// TIA Portal V20 export
// export: Created 2025-12-01T14:56:59.921487Z, ExportSetting None, DisplayName Totally Integrated Automation Portal, DisplayVersion V20 Update 3, DisplayName TIA Portal Openness, DisplayVersion V20 Update 3, DisplayName TIA Portal Version Control Interface, DisplayVersion V20 Update 3, DisplayName STEP 7 Professional, DisplayVersion V20 Update 3, DisplayName STEP 7 Safety, DisplayVersion V20 Update 2, DisplayName WinCC Basic/Comfort/Advanced, DisplayVersion V20 Update 3, DisplayName WinCC Professional, DisplayVersion V20 Update 3, DisplayName WinCC Unified, DisplayVersion V20 Update 3
FUNCTION "FC425_TL_Sep_Salida" : Void   // FC425, LAD
{ S7_Optimized_Access := 'FALSE' }
AUTHOR : TLigero
NAME : 20190131
VERSION : 3.3
// ////////////////////////////
// Modificada 27-11-2012
// Separación salida entre culo de primera caja y cara de la segunda para distanci 
// kte mayor flujo con tamaños diferentes de cajas
// ////////////////////////////
// stored: AutoNumber false, SetENOAutomatically false
   VAR_INPUT
      Mesa : UInt;
      En_Tension : Bool;
      PhsMx : Bool;
      Termico_Tx : Bool;
      Avance_Tx : Bool;
      Modo_Pasoapaso_Tx : Bool;
      AVTF_MAnt_Mx : Bool;
      PTF_Mx_MSig : Bool;
      NXT_Avance : Bool;
      V_CNT_pHsMx : UDInt;
      V_Paro : UDInt;
      V_Separacion : UDInt;
      V_Caja_Max : UDInt;
      V_TOut_Tx_Mx : UDInt;
      V_Acumulacion : UDInt;
   END_VAR
   VAR_OUTPUT
      PTF_MAnt_Mx : Bool;
      AVTF_Mx_MSig : Bool;
   END_VAR
   VAR_IN_OUT
      NXT_Descarga_Act : Bool;
      Carga_Activa_Tx : Bool;
      MAUX_FN_AVTF : Bool;
      Mem_CNT_Tmp_PRES : Bool;
      Mem_CNT_Tmp_Paro_Tx : Bool;
      Mem_CNT_Acumulacion : Bool;
   END_VAR
   VAR_TEMP
      CNT_Sep : Word;
      CNT_Sep_Int : Int;
      CNT_Sep_FORZ_Sep : Int;
      Aux_Parar : Bool;
      Mem_CNT_Separacion : Bool;
      ok_tension : Bool;
      mem_atasco : Bool;
   END_VAR
   VAR_TEMP   // added for the SCL form of the ladder/FBD networks
      _w1 : Bool;
   END_VAR
BEGIN

REGION Network 1: Marca General Error
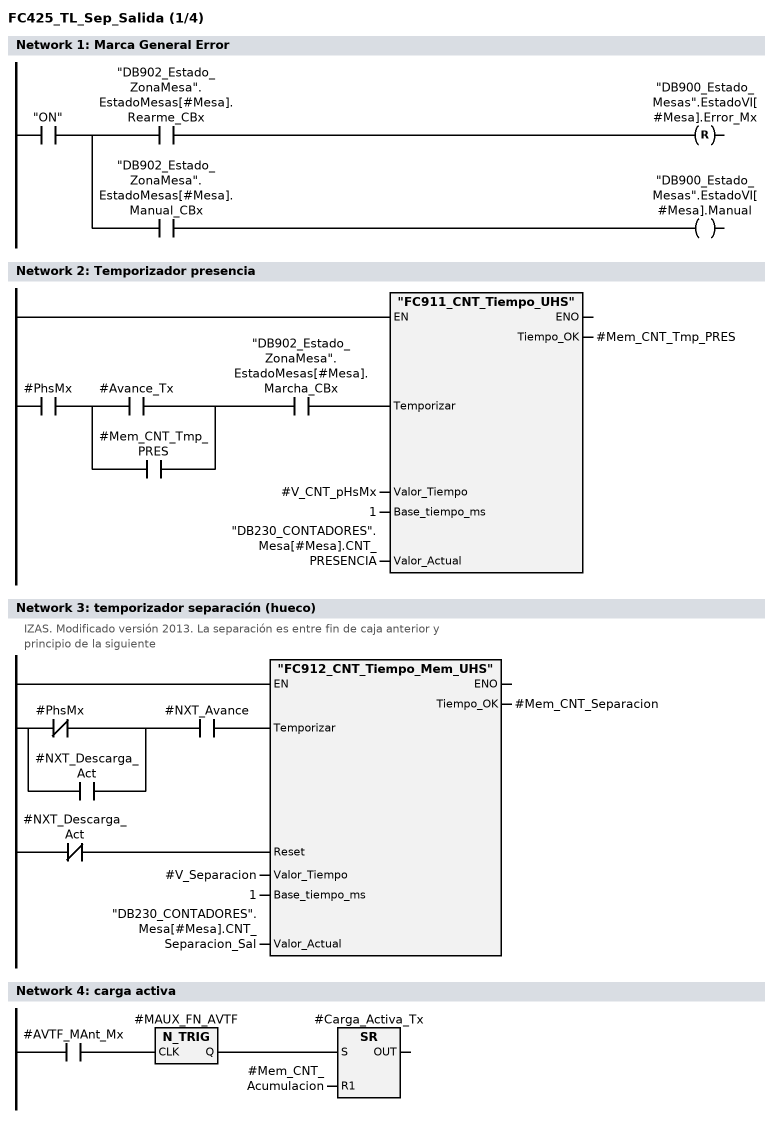
   RUNG wire#powerrail
      Contact( "ON" )
      wire#w1
      Contact( "DB902_Estado_ZonaMesa".EstadoMesas[#Mesa].Rearme_CBx )
      R_Coil( "DB900_Estado_Mesas".EstadoVI[#Mesa].Error_Mx )
   END_RUNG
   RUNG wire#w1
      Contact( "DB902_Estado_ZonaMesa".EstadoMesas[#Mesa].Manual_CBx )
      Coil( "DB900_Estado_Mesas".EstadoVI[#Mesa].Manual )
   END_RUNG
   // the same network as SCL:
   IF "ON" AND "DB902_Estado_ZonaMesa".EstadoMesas[#Mesa].Rearme_CBx THEN
       "DB900_Estado_Mesas".EstadoVI[#Mesa].Error_Mx := FALSE;
   END_IF;
   "DB900_Estado_Mesas".EstadoVI[#Mesa].Manual := "ON" AND "DB902_Estado_ZonaMesa".EstadoMesas[#Mesa].Manual_CBx;
END_REGION

REGION Network 2: Temporizador presencia
   RUNG wire#powerrail
      "FC911_CNT_Tiempo_UHS"(Temporizar := wire#w3, Valor_Tiempo := #V_CNT_pHsMx, Base_tiempo_ms := 1, Valor_Actual := "DB230_CONTADORES".Mesa[#Mesa].CNT_PRESENCIA, Tiempo_OK => #Mem_CNT_Tmp_PRES)
   END_RUNG
   RUNG wire#powerrail
      Contact( #PhsMx )
      wire#w1
      Contact( #Avance_Tx )
      wire#w2
      Contact( "DB902_Estado_ZonaMesa".EstadoMesas[#Mesa].Marcha_CBx )
   END_RUNG wire#w3
   RUNG wire#w1
      Contact( #Mem_CNT_Tmp_PRES )
   END_RUNG wire#w2
   // the same network as SCL:
   "FC911_CNT_Tiempo_UHS"(Temporizar := #PhsMx AND (#Avance_Tx OR #Mem_CNT_Tmp_PRES) AND "DB902_Estado_ZonaMesa".EstadoMesas[#Mesa].Marcha_CBx,
                          Valor_Tiempo := #V_CNT_pHsMx,
                          Base_tiempo_ms := 1,
                          Valor_Actual := "DB230_CONTADORES".Mesa[#Mesa].CNT_PRESENCIA,
                          Tiempo_OK => #Mem_CNT_Tmp_PRES);
END_REGION

REGION Network 3: temporizador separación (hueco)
   // IZAS. Modificado versión 2013. La separación es entre fin de caja anterior y 
   // principio de la siguiente
   RUNG wire#powerrail
      "FC912_CNT_Tiempo_Mem_UHS"(Temporizar := wire#w2, Reset := wire#w3, Valor_Tiempo := #V_Separacion, Base_tiempo_ms := 1, Valor_Actual := "DB230_CONTADORES".Mesa[#Mesa].CNT_Separacion_Sal, Tiempo_OK => #Mem_CNT_Separacion)
   END_RUNG
   RUNG wire#powerrail
      I_Contact( #PhsMx )
      wire#w1
      Contact( #NXT_Avance )
   END_RUNG wire#w2
   RUNG wire#powerrail
      Contact( #NXT_Descarga_Act )
   END_RUNG wire#w1
   RUNG wire#powerrail
      I_Contact( #NXT_Descarga_Act )
   END_RUNG wire#w3
   // the same network as SCL:
   "FC912_CNT_Tiempo_Mem_UHS"(Temporizar := (NOT #PhsMx OR #NXT_Descarga_Act) AND #NXT_Avance,
                           Reset := NOT #NXT_Descarga_Act,
                           Valor_Tiempo := #V_Separacion,
                           Base_tiempo_ms := 1,
                           Valor_Actual := "DB230_CONTADORES".Mesa[#Mesa].CNT_Separacion_Sal,
                           Tiempo_OK => #Mem_CNT_Separacion);
END_REGION

REGION Network 4: carga activa
   RUNG wire#powerrail
      Contact( #AVTF_MAnt_Mx )
      N_Trig( #MAUX_FN_AVTF )
      S_SR(operand := #Carga_Activa_Tx, r1 := #Mem_CNT_Acumulacion)
   END_RUNG
   // the same network as SCL:
   #_w1 := NOT #AVTF_MAnt_Mx AND #MAUX_FN_AVTF;   // falling edge
   #MAUX_FN_AVTF := #AVTF_MAnt_Mx;
   IF #_w1 THEN
       #Carga_Activa_Tx := TRUE;   // SR flip-flop
   END_IF;
   IF #Mem_CNT_Acumulacion THEN #Carga_Activa_Tx := FALSE; END_IF;
END_REGION

REGION Network 5: Temporizador acumulacion
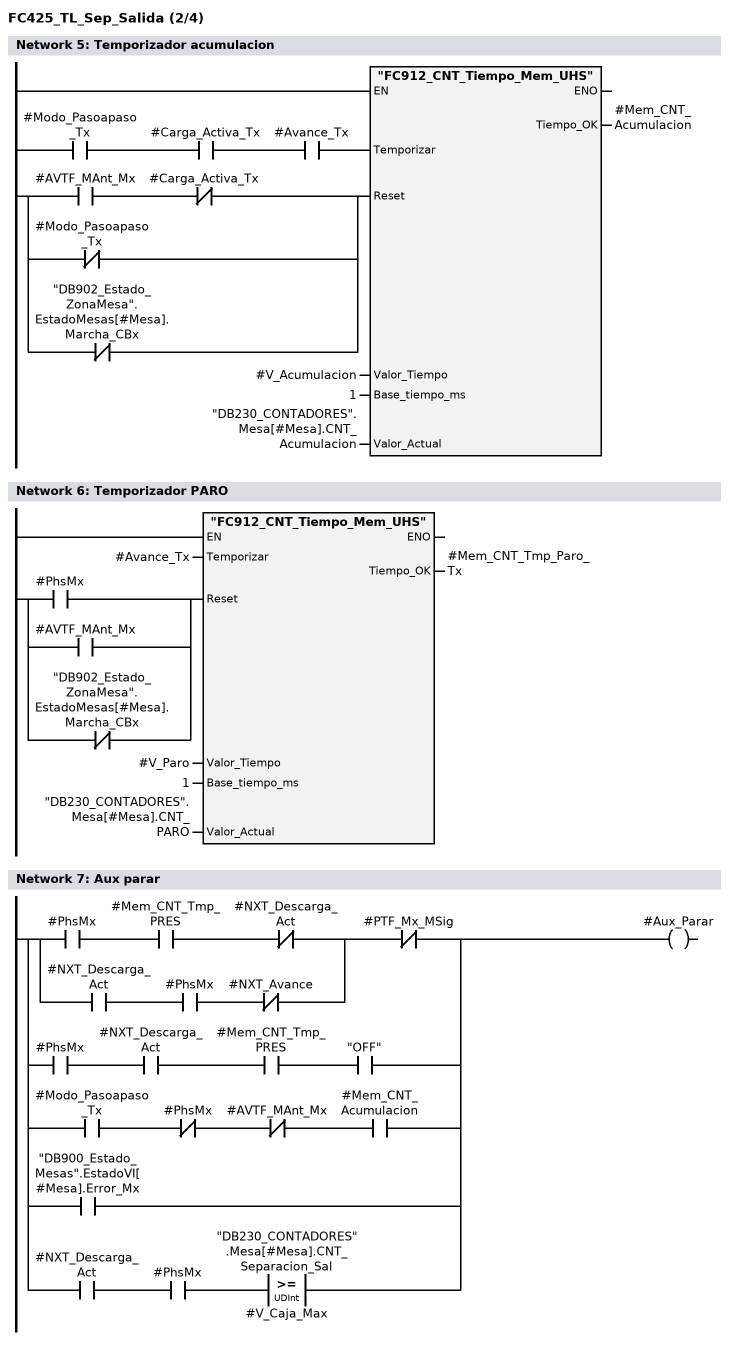
   RUNG wire#powerrail
      "FC912_CNT_Tiempo_Mem_UHS"(Temporizar := wire#w1, Reset := wire#w2, Valor_Tiempo := #V_Acumulacion, Base_tiempo_ms := 1, Valor_Actual := "DB230_CONTADORES".Mesa[#Mesa].CNT_Acumulacion, Tiempo_OK => #Mem_CNT_Acumulacion)
   END_RUNG
   RUNG wire#powerrail
      Contact( #Modo_Pasoapaso_Tx )
      Contact( #Carga_Activa_Tx )
      Contact( #Avance_Tx )
   END_RUNG wire#w1
   RUNG wire#powerrail
      Contact( #AVTF_MAnt_Mx )
      I_Contact( #Carga_Activa_Tx )
   END_RUNG wire#w2
   RUNG wire#powerrail
      I_Contact( #Modo_Pasoapaso_Tx )
   END_RUNG wire#w2
   RUNG wire#powerrail
      I_Contact( "DB902_Estado_ZonaMesa".EstadoMesas[#Mesa].Marcha_CBx )
   END_RUNG wire#w2
   // the same network as SCL:
   "FC912_CNT_Tiempo_Mem_UHS"(Temporizar := #Modo_Pasoapaso_Tx AND #Carga_Activa_Tx AND #Avance_Tx,
                           Reset := (#AVTF_MAnt_Mx AND NOT #Carga_Activa_Tx) OR NOT #Modo_Pasoapaso_Tx OR NOT "DB902_Estado_ZonaMesa".EstadoMesas[#Mesa].Marcha_CBx,
                           Valor_Tiempo := #V_Acumulacion,
                           Base_tiempo_ms := 1,
                           Valor_Actual := "DB230_CONTADORES".Mesa[#Mesa].CNT_Acumulacion,
                           Tiempo_OK => #Mem_CNT_Acumulacion);
END_REGION

REGION Network 6: Temporizador PARO
   RUNG wire#powerrail
      "FC912_CNT_Tiempo_Mem_UHS"(Reset := wire#w1, Temporizar := #Avance_Tx, Valor_Tiempo := #V_Paro, Base_tiempo_ms := 1, Valor_Actual := "DB230_CONTADORES".Mesa[#Mesa].CNT_PARO, Tiempo_OK => #Mem_CNT_Tmp_Paro_Tx)
   END_RUNG
   RUNG wire#powerrail
      Contact( #PhsMx )
   END_RUNG wire#w1
   RUNG wire#powerrail
      Contact( #AVTF_MAnt_Mx )
   END_RUNG wire#w1
   RUNG wire#powerrail
      I_Contact( "DB902_Estado_ZonaMesa".EstadoMesas[#Mesa].Marcha_CBx )
   END_RUNG wire#w1
   // the same network as SCL:
   "FC912_CNT_Tiempo_Mem_UHS"(Temporizar := #Avance_Tx,
                           Reset := #PhsMx OR #AVTF_MAnt_Mx OR NOT "DB902_Estado_ZonaMesa".EstadoMesas[#Mesa].Marcha_CBx,
                           Valor_Tiempo := #V_Paro,
                           Base_tiempo_ms := 1,
                           Valor_Actual := "DB230_CONTADORES".Mesa[#Mesa].CNT_PARO,
                           Tiempo_OK => #Mem_CNT_Tmp_Paro_Tx);
END_REGION

REGION Network 7: Aux parar
   RUNG wire#powerrail
      Contact( #PhsMx )
      Contact( #Mem_CNT_Tmp_PRES )
      I_Contact( #NXT_Descarga_Act )
      wire#w1
      I_Contact( #PTF_Mx_MSig )
      wire#w2
      Coil( #Aux_Parar )
   END_RUNG
   RUNG wire#powerrail
      Contact( #NXT_Descarga_Act )
      Contact( #PhsMx )
      I_Contact( #NXT_Avance )
   END_RUNG wire#w1
   RUNG wire#powerrail
      Contact( #PhsMx )
      Contact( #NXT_Descarga_Act )
      Contact( #Mem_CNT_Tmp_PRES )
      Contact( "OFF" )
   END_RUNG wire#w2
   RUNG wire#powerrail
      Contact( #Modo_Pasoapaso_Tx )
      I_Contact( #PhsMx )
      I_Contact( #AVTF_MAnt_Mx )
      Contact( #Mem_CNT_Acumulacion )
   END_RUNG wire#w2
   RUNG wire#powerrail
      Contact( "DB900_Estado_Mesas".EstadoVI[#Mesa].Error_Mx )
   END_RUNG wire#w2
   RUNG wire#powerrail
      Contact( #NXT_Descarga_Act )
      Contact( #PhsMx )
      { S7_Templates := "SrcType := UDInt" } GE_Contact(in1 := "DB230_CONTADORES".Mesa[#Mesa].CNT_Separacion_Sal, in2 := #V_Caja_Max)
   END_RUNG wire#w2
   // the same network as SCL:
   #Aux_Parar := (((#PhsMx AND #Mem_CNT_Tmp_PRES AND NOT #NXT_Descarga_Act) OR (#NXT_Descarga_Act AND #PhsMx AND NOT #NXT_Avance)) AND NOT #PTF_Mx_MSig) OR (#PhsMx AND #NXT_Descarga_Act AND #Mem_CNT_Tmp_PRES AND "OFF") OR (#Modo_Pasoapaso_Tx AND NOT #PhsMx AND NOT #AVTF_MAnt_Mx AND #Mem_CNT_Acumulacion) OR "DB900_Estado_Mesas".EstadoVI[#Mesa].Error_Mx OR (#NXT_Descarga_Act AND #PhsMx AND ("DB230_CONTADORES".Mesa[#Mesa].CNT_Separacion_Sal >= #V_Caja_Max));
END_REGION

REGION Network 8: NXT descarga activa
   // modificado despues de hablar con carlos.
   // Antes el reseteo era con la variable del contador negada
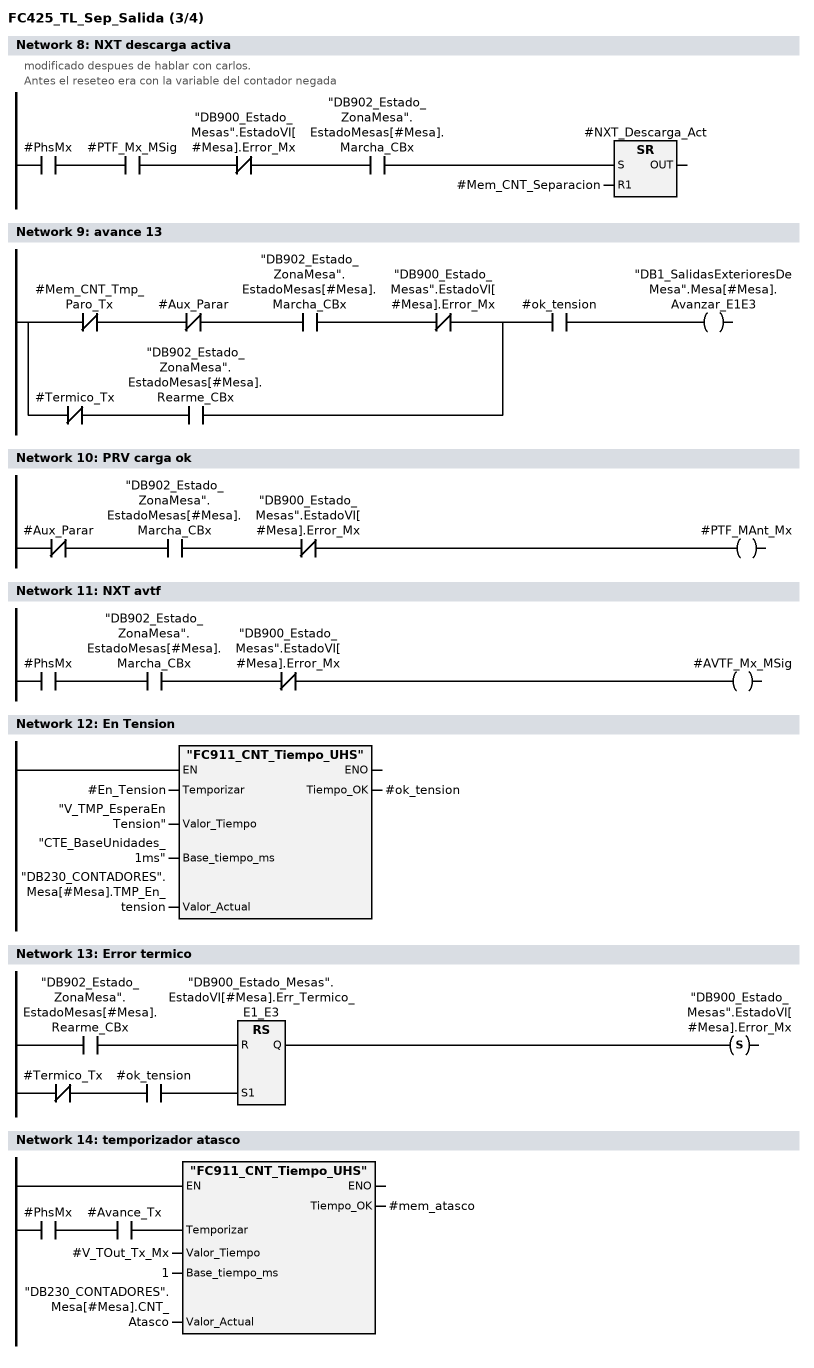
   RUNG wire#powerrail
      Contact( #PhsMx )
      Contact( #PTF_Mx_MSig )
      I_Contact( "DB900_Estado_Mesas".EstadoVI[#Mesa].Error_Mx )
      Contact( "DB902_Estado_ZonaMesa".EstadoMesas[#Mesa].Marcha_CBx )
      S_SR(operand := #NXT_Descarga_Act, r1 := #Mem_CNT_Separacion)
   END_RUNG
   // the same network as SCL:
   IF #PhsMx AND #PTF_Mx_MSig AND NOT "DB900_Estado_Mesas".EstadoVI[#Mesa].Error_Mx AND "DB902_Estado_ZonaMesa".EstadoMesas[#Mesa].Marcha_CBx THEN
       #NXT_Descarga_Act := TRUE;   // SR flip-flop
   END_IF;
   IF #Mem_CNT_Separacion THEN #NXT_Descarga_Act := FALSE; END_IF;
END_REGION

REGION Network 9: avance 13
   RUNG wire#powerrail
      I_Contact( #Mem_CNT_Tmp_Paro_Tx )
      I_Contact( #Aux_Parar )
      Contact( "DB902_Estado_ZonaMesa".EstadoMesas[#Mesa].Marcha_CBx )
      I_Contact( "DB900_Estado_Mesas".EstadoVI[#Mesa].Error_Mx )
      wire#w1
      Contact( #ok_tension )
      Coil( "DB1_SalidasExterioresDeMesa".Mesa[#Mesa].Avanzar_E1E3 )
   END_RUNG
   RUNG wire#powerrail
      I_Contact( #Termico_Tx )
      Contact( "DB902_Estado_ZonaMesa".EstadoMesas[#Mesa].Rearme_CBx )
   END_RUNG wire#w1
   // the same network as SCL:
   "DB1_SalidasExterioresDeMesa".Mesa[#Mesa].Avanzar_E1E3 := ((NOT #Mem_CNT_Tmp_Paro_Tx AND NOT #Aux_Parar AND "DB902_Estado_ZonaMesa".EstadoMesas[#Mesa].Marcha_CBx AND NOT "DB900_Estado_Mesas".EstadoVI[#Mesa].Error_Mx) OR (NOT #Termico_Tx AND "DB902_Estado_ZonaMesa".EstadoMesas[#Mesa].Rearme_CBx)) AND #ok_tension;
END_REGION

REGION Network 10: PRV carga ok
   RUNG wire#powerrail
      I_Contact( #Aux_Parar )
      Contact( "DB902_Estado_ZonaMesa".EstadoMesas[#Mesa].Marcha_CBx )
      I_Contact( "DB900_Estado_Mesas".EstadoVI[#Mesa].Error_Mx )
      Coil( #PTF_MAnt_Mx )
   END_RUNG
   // the same network as SCL:
   #PTF_MAnt_Mx := NOT #Aux_Parar AND "DB902_Estado_ZonaMesa".EstadoMesas[#Mesa].Marcha_CBx AND NOT "DB900_Estado_Mesas".EstadoVI[#Mesa].Error_Mx;
END_REGION

REGION Network 11: NXT avtf
   RUNG wire#powerrail
      Contact( #PhsMx )
      Contact( "DB902_Estado_ZonaMesa".EstadoMesas[#Mesa].Marcha_CBx )
      I_Contact( "DB900_Estado_Mesas".EstadoVI[#Mesa].Error_Mx )
      Coil( #AVTF_Mx_MSig )
   END_RUNG
   // the same network as SCL:
   #AVTF_Mx_MSig := #PhsMx AND "DB902_Estado_ZonaMesa".EstadoMesas[#Mesa].Marcha_CBx AND NOT "DB900_Estado_Mesas".EstadoVI[#Mesa].Error_Mx;
END_REGION

REGION Network 12: En Tension
   RUNG wire#powerrail
      "FC911_CNT_Tiempo_UHS"(Temporizar := #En_Tension, Valor_Tiempo := "V_TMP_EsperaEnTension", Base_tiempo_ms := "CTE_BaseUnidades_1ms", Valor_Actual := "DB230_CONTADORES".Mesa[#Mesa].TMP_En_tension, Tiempo_OK => #ok_tension)
   END_RUNG
   // the same network as SCL:
   "FC911_CNT_Tiempo_UHS"(Temporizar := #En_Tension,
                          Valor_Tiempo := "V_TMP_EsperaEnTension",
                          Base_tiempo_ms := "CTE_BaseUnidades_1ms",
                          Valor_Actual := "DB230_CONTADORES".Mesa[#Mesa].TMP_En_tension,
                          Tiempo_OK => #ok_tension);
END_REGION

REGION Network 13: Error termico
   RUNG wire#powerrail
      Contact( "DB902_Estado_ZonaMesa".EstadoMesas[#Mesa].Rearme_CBx )
      S_RS(operand := "DB900_Estado_Mesas".EstadoVI[#Mesa].Err_Termico_E1_E3, s1 := wire#w1)
      S_Coil( "DB900_Estado_Mesas".EstadoVI[#Mesa].Error_Mx )
   END_RUNG
   RUNG wire#powerrail
      I_Contact( #Termico_Tx )
      Contact( #ok_tension )
   END_RUNG wire#w1
   // the same network as SCL:
   IF "DB902_Estado_ZonaMesa".EstadoMesas[#Mesa].Rearme_CBx THEN
       "DB900_Estado_Mesas".EstadoVI[#Mesa].Err_Termico_E1_E3 := FALSE;   // RS flip-flop
   END_IF;
   IF NOT #Termico_Tx AND #ok_tension THEN
       "DB900_Estado_Mesas".EstadoVI[#Mesa].Err_Termico_E1_E3 := TRUE;
   END_IF;
   IF "DB900_Estado_Mesas".EstadoVI[#Mesa].Err_Termico_E1_E3 THEN
       "DB900_Estado_Mesas".EstadoVI[#Mesa].Error_Mx := TRUE;
   END_IF;
END_REGION

REGION Network 14: temporizador atasco
   RUNG wire#powerrail
      "FC911_CNT_Tiempo_UHS"(Temporizar := wire#w1, Valor_Tiempo := #V_TOut_Tx_Mx, Base_tiempo_ms := 1, Valor_Actual := "DB230_CONTADORES".Mesa[#Mesa].CNT_Atasco, Tiempo_OK => #mem_atasco)
   END_RUNG
   RUNG wire#powerrail
      Contact( #PhsMx )
      Contact( #Avance_Tx )
   END_RUNG wire#w1
   // the same network as SCL:
   "FC911_CNT_Tiempo_UHS"(Temporizar := #PhsMx AND #Avance_Tx,
                          Valor_Tiempo := #V_TOut_Tx_Mx,
                          Base_tiempo_ms := 1,
                          Valor_Actual := "DB230_CONTADORES".Mesa[#Mesa].CNT_Atasco,
                          Tiempo_OK => #mem_atasco);
END_REGION

REGION Network 15: Error atasco
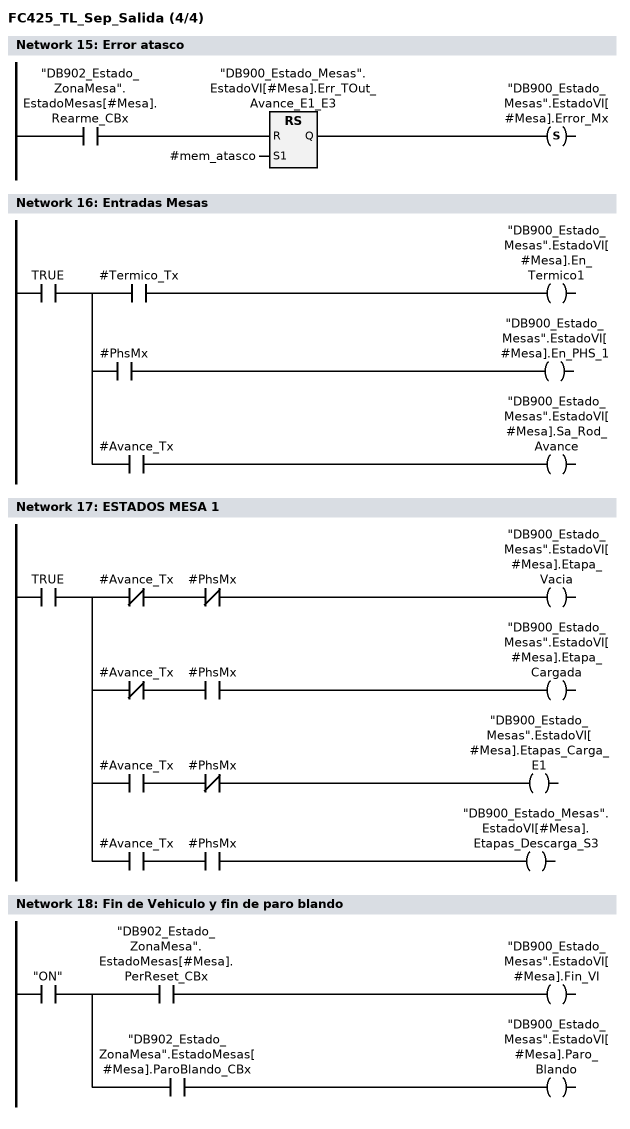
   RUNG wire#powerrail
      Contact( "DB902_Estado_ZonaMesa".EstadoMesas[#Mesa].Rearme_CBx )
      S_RS(operand := "DB900_Estado_Mesas".EstadoVI[#Mesa].Err_TOut_Avance_E1_E3, s1 := #mem_atasco)
      S_Coil( "DB900_Estado_Mesas".EstadoVI[#Mesa].Error_Mx )
   END_RUNG
   // the same network as SCL:
   IF "DB902_Estado_ZonaMesa".EstadoMesas[#Mesa].Rearme_CBx THEN
       "DB900_Estado_Mesas".EstadoVI[#Mesa].Err_TOut_Avance_E1_E3 := FALSE;   // RS flip-flop
   END_IF;
   IF #mem_atasco THEN "DB900_Estado_Mesas".EstadoVI[#Mesa].Err_TOut_Avance_E1_E3 := TRUE; END_IF;
   IF "DB900_Estado_Mesas".EstadoVI[#Mesa].Err_TOut_Avance_E1_E3 THEN
       "DB900_Estado_Mesas".EstadoVI[#Mesa].Error_Mx := TRUE;
   END_IF;
END_REGION

REGION Network 16: Entradas Mesas
   RUNG wire#powerrail
      Contact( TRUE )
      wire#w1
      Contact( #Termico_Tx )
      Coil( "DB900_Estado_Mesas".EstadoVI[#Mesa].En_Termico1 )
   END_RUNG
   RUNG wire#w1
      Contact( #PhsMx )
      Coil( "DB900_Estado_Mesas".EstadoVI[#Mesa].En_PHS_1 )
   END_RUNG
   RUNG wire#w1
      Contact( #Avance_Tx )
      Coil( "DB900_Estado_Mesas".EstadoVI[#Mesa].Sa_Rod_Avance )
   END_RUNG
   // the same network as SCL:
   "DB900_Estado_Mesas".EstadoVI[#Mesa].En_Termico1 := TRUE AND #Termico_Tx;
   "DB900_Estado_Mesas".EstadoVI[#Mesa].En_PHS_1 := TRUE AND #PhsMx;
   "DB900_Estado_Mesas".EstadoVI[#Mesa].Sa_Rod_Avance := TRUE AND #Avance_Tx;
END_REGION

REGION Network 17: ESTADOS MESA 1
   RUNG wire#powerrail
      Contact( TRUE )
      wire#w1
      I_Contact( #Avance_Tx )
      I_Contact( #PhsMx )
      Coil( "DB900_Estado_Mesas".EstadoVI[#Mesa].Etapa_Vacia )
   END_RUNG
   RUNG wire#w1
      I_Contact( #Avance_Tx )
      Contact( #PhsMx )
      Coil( "DB900_Estado_Mesas".EstadoVI[#Mesa].Etapa_Cargada )
   END_RUNG
   RUNG wire#w1
      Contact( #Avance_Tx )
      I_Contact( #PhsMx )
      Coil( "DB900_Estado_Mesas".EstadoVI[#Mesa].Etapas_Carga_E1 )
   END_RUNG
   RUNG wire#w1
      Contact( #Avance_Tx )
      Contact( #PhsMx )
      Coil( "DB900_Estado_Mesas".EstadoVI[#Mesa].Etapas_Descarga_S3 )
   END_RUNG
   // the same network as SCL:
   "DB900_Estado_Mesas".EstadoVI[#Mesa].Etapa_Vacia := TRUE AND NOT #Avance_Tx AND NOT #PhsMx;
   "DB900_Estado_Mesas".EstadoVI[#Mesa].Etapa_Cargada := TRUE AND NOT #Avance_Tx AND #PhsMx;
   "DB900_Estado_Mesas".EstadoVI[#Mesa].Etapas_Carga_E1 := TRUE AND #Avance_Tx AND NOT #PhsMx;
   "DB900_Estado_Mesas".EstadoVI[#Mesa].Etapas_Descarga_S3 := TRUE AND #Avance_Tx AND #PhsMx;
END_REGION

REGION Network 18: Fin de Vehiculo y fin de paro blando
   RUNG wire#powerrail
      Contact( "ON" )
      wire#w1
      Contact( "DB902_Estado_ZonaMesa".EstadoMesas[#Mesa].PerReset_CBx )
      Coil( "DB900_Estado_Mesas".EstadoVI[#Mesa].Fin_VI )
   END_RUNG
   RUNG wire#w1
      Contact( "DB902_Estado_ZonaMesa".EstadoMesas[#Mesa].ParoBlando_CBx )
      Coil( "DB900_Estado_Mesas".EstadoVI[#Mesa].Paro_Blando )
   END_RUNG
   // the same network as SCL:
   "DB900_Estado_Mesas".EstadoVI[#Mesa].Fin_VI := "ON" AND "DB902_Estado_ZonaMesa".EstadoMesas[#Mesa].PerReset_CBx;
   "DB900_Estado_Mesas".EstadoVI[#Mesa].Paro_Blando := "ON" AND "DB902_Estado_ZonaMesa".EstadoMesas[#Mesa].ParoBlando_CBx;
END_REGION
END_FUNCTION
